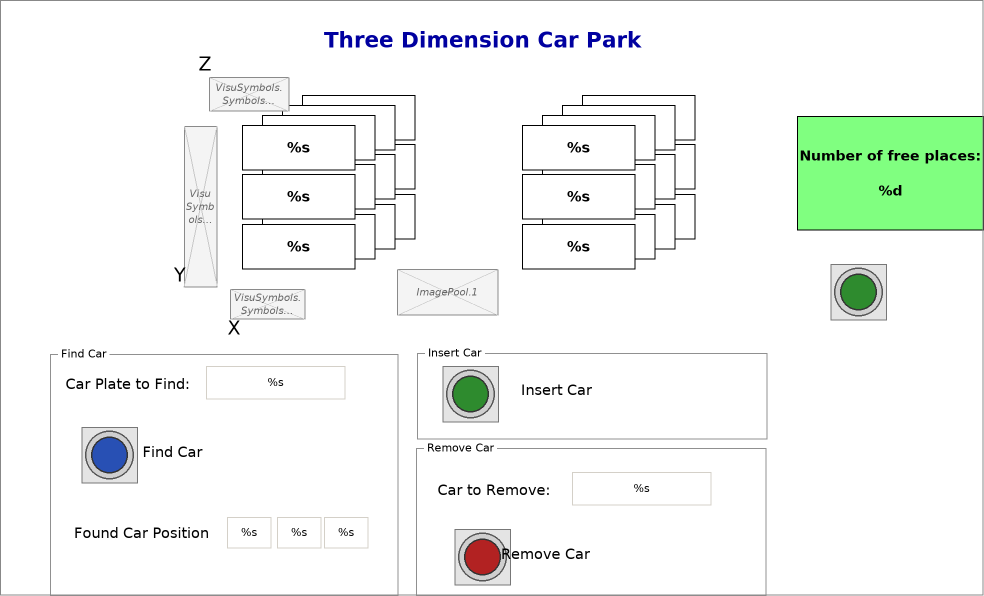
VISUALIZATION Visualization  // 984x596
    Rectangle (302,95 113x45), "%s", text variable: MAIN.CarPark[1,3,4], colour toggle: MAIN.CarPark[1,3,4] <> ''
    Rectangle (302,194 113x45), "%s", text variable: MAIN.CarPark[1,1,4], colour toggle: MAIN.CarPark[1,1,4] <> ''
    Rectangle (302,144 113x45), "%s", text variable: MAIN.CarPark[1,2,4], colour toggle: MAIN.CarPark[1,2,4] <> ''
    Rectangle (282,204 113x45), "%s", text variable: MAIN.CarPark[1,1,3], colour toggle: MAIN.CarPark[1,1,3] <> ''
    Rectangle (282,154 113x45), "%s", text variable: MAIN.CarPark[1,2,3], colour toggle: MAIN.CarPark[1,2,3] <> ''
    Rectangle (282,105 113x45), "%s", text variable: MAIN.CarPark[1,3,3], colour toggle: MAIN.CarPark[1,3,3] <> ''
    Rectangle (262,115 113x45), "%s", text variable: MAIN.CarPark[1,3,2], colour toggle: MAIN.CarPark[1,3,2] <> ''
    Rectangle (262,164 113x45), "%s", text variable: MAIN.CarPark[1,2,2], colour toggle: MAIN.CarPark[1,2,2] <> ''
    Rectangle (262,214 113x45), "%s", text variable: MAIN.CarPark[1,1,2], colour toggle: MAIN.CarPark[1,1,2] <> ''
    Rectangle (242,224 113x45), "%s", text variable: MAIN.CarPark[1,1,1], colour toggle: MAIN.CarPark[1,1,1] <> ''
    Rectangle (242,174 113x45), "%s", text variable: MAIN.CarPark[1,2,1], colour toggle: MAIN.CarPark[1,2,1] <> ''
    Rectangle (242,125 113x45), "%s", text variable: MAIN.CarPark[1,3,1], colour toggle: MAIN.CarPark[1,3,1] <> ''
    Rectangle (582,95 113x45), "%s", text variable: MAIN.CarPark[2,3,4], colour toggle: MAIN.CarPark[2,3,4] <> ''
    Rectangle (582,194 113x45), "%s", text variable: MAIN.CarPark[2,1,4], colour toggle: MAIN.CarPark[2,1,4] <> ''
    Rectangle (582,144 113x45), "%s", text variable: MAIN.CarPark[2,2,4], colour toggle: MAIN.CarPark[2,2,4] <> ''
    Rectangle (562,204 113x45), "%s", text variable: MAIN.CarPark[2,1,3], colour toggle: MAIN.CarPark[2,1,3] <> ''
    Rectangle (562,154 113x45), "%s", text variable: MAIN.CarPark[2,2,3], colour toggle: MAIN.CarPark[2,2,3] <> ''
    Rectangle (562,105 113x45), "%s", text variable: MAIN.CarPark[2,3,3], colour toggle: MAIN.CarPark[2,3,3] <> ''
    Rectangle (542,115 113x45), "%s", text variable: MAIN.CarPark[2,3,2], colour toggle: MAIN.CarPark[2,3,2] <> ''
    Rectangle (542,164 113x45), "%s", text variable: MAIN.CarPark[2,2,2], colour toggle: MAIN.CarPark[2,2,2] <> ''
    Rectangle (542,214 113x45), "%s", text variable: MAIN.CarPark[2,1,2], colour toggle: MAIN.CarPark[2,1,2] <> ''
    Rectangle (522,224 113x45), "%s", text variable: MAIN.CarPark[2,1,1], colour toggle: MAIN.CarPark[2,1,1] <> ''
    Rectangle (522,174 113x45), "%s", text variable: MAIN.CarPark[2,2,1], colour toggle: MAIN.CarPark[2,2,1] <> ''
    Rectangle (522,125 113x45), "%s", text variable: MAIN.CarPark[2,3,1], colour toggle: MAIN.CarPark[2,3,1] <> ''
    Label (319,22 328x36), "Three Dimension Car Park"
    GroupBox (50,346 348x250), "Find Car"
        Label (3,20 150x36), "Car Plate to Find:"
        Textfield (156,20 139x33), "%s", tooltip "Plate to find", text variable: MAIN.PlateToFind
            OnMouseClick: write the text variable via Edit
        PushSwitch (20,81 79x56), tooltip "Find Car", variable: MAIN.FindCar, behaviour: TAP, style: Switch-PushSwitch-Blue
        Label (72,88 101x36), "Find Car"
        Label (9,169 165x36), "Found Car Position"
        Textfield (177,171 44x31), "%s", tooltip "Plate to find", text variable: MAIN.CarFoundPos.X
            OnMouseClick: write the text variable via Edit
        Textfield (227,171 44x31), "%s", tooltip "Plate to find", text variable: MAIN.CarFoundPos.Y
            OnMouseClick: write the text variable via Edit
        Textfield (274,171 44x31), "%s", tooltip "Plate to find", text variable: MAIN.CarFoundPos.Z
            OnMouseClick: write the text variable via Edit
        PushSwitch (769,-82 79x56), tooltip "Find Car", variable: MAIN.FindCar, behaviour: TAP, style: Switch-PushSwitch-Green
    Rectangle (797,116 187x114), "Number of free places: %d", text variable: MAIN.FreePlaces
    GroupBox (416,440 350x156), "Remove Car"
        Label (3,32 150x36), "Car to Remove:"
        Textfield (156,32 139x33), "%s", tooltip "Car to remove", text variable: MAIN.CarToRemove
            OnMouseClick: write the text variable via Edit
        PushSwitch (27,89 79x56), tooltip "Remove Car", variable: MAIN.RemoveCar, behaviour: TAP, style: Switch-PushSwitch-Red
        Label (79,96 101x36), "Remove Car"
    GroupBox (417,345 350x94), "Insert Car"
        PushSwitch (14,21 79x56), tooltip "Insert Car", variable: MAIN.InsertCar, behaviour: TAP, style: Switch-PushSwitch-Green
        Label (89,27 101x36), "Insert Car"
    Image (397,269 101x46), image: ImagePool.1
    Image (230,289 75x30), image: VisuSymbols.Symbols.ArrowBoldRight
    Image (184,126 33x161), image: VisuSymbols.Symbols.ArrowBoldUp
    Image (209,77 80x34), image: VisuSymbols.Symbols.ArrowBoldRightUp
    Label (214,310 40x36), "X"
    Label (160,257 40x36), "Y"
    Label (185,46 40x36), "Z"
END_VISUALIZATION

(* stored: Version 1.1.0.1, ProductVersion 3.1.4024.15
   Visu Visualization: Id {062b7834-b7fb-4631-b721-dcb9f809d15d} *)
